TYPE
    StatusCam :
    STRUCT
        Error                : BOOL;
        Warning              : BOOL;
        CurrentValueProperty : BOOL;
        ErrorId              : UINT;
    END_STRUCT
END_TYPE

(* stored: Version 1.1.0.1, ProductVersion 3.1.4024.12
   DUT StatusCam: Id {b6ee1a61-02fb-4d9b-9af8-a94c50c9b414} *)
